_CFC_ (* Continuous Function Chart, elements in execution order *)
(* 3s *)
(* 3s *)
(* 90s *)
(* 1s *)
#0 AND(#3.Q, #6.Q)
#1 INT_TO_TIME(SHU6_PV1_ZADER_VPDS_OTSUT)
#2 MUL(#1, 1000)
#3 TON_PDS3:TON(IN: NOT SHU6_PV1_1PDS5_DI4, PT: #2)
#4 INT_TO_TIME(SHU6_PV1_ZADER_VPDS_RABOTA)
#5 MUL(#4, 1000)
#6 TON_ReRab:TON(IN: SHU6_PV1_UST_RE_RABOTA, PT: #5)
#7 INT_TO_TIME(SHU6_PV1_ZADER_M_VKL)
#8 MUL(#7, 1000)
#9 TON_MVKL_MV1:TON(IN: SHU6_PV1_MV1_DO3_VKL, PT: #8)
#10 INT_TO_TIME(SHU6_PV1_ZADER_M_A)
#11 MUL(#10, 1000)
#12 TON_AVT_MV1:TON(IN: SHU6_PV1_YAMV1_DI7_A, PT: #11)
#13 AND(#0, SHU6_PV1_MV1_B30, #9.Q, #12.Q)
#14 SR_NP_MV1:SR(SET1: #13, RESET: SHU6_PV1_SB)
#15 SHU6_PV1_Z_NETP_MV1 <= #14.Q1
_END_CFC_
(* the same logic as Structured Text *)
(* 3s *)
(* 3s *)
(* 90s *)
(* 1s *)
_t70 := TON_PDS3.Q AND TON_ReRab.Q;
TON_PDS3(IN := NOT SHU6_PV1_1PDS5_DI4, PT := INT_TO_TIME(SHU6_PV1_ZADER_VPDS_OTSUT) * 1000);
TON_ReRab(IN := SHU6_PV1_UST_RE_RABOTA, PT := INT_TO_TIME(SHU6_PV1_ZADER_VPDS_RABOTA) * 1000);
TON_MVKL_MV1(IN := SHU6_PV1_MV1_DO3_VKL, PT := INT_TO_TIME(SHU6_PV1_ZADER_M_VKL) * 1000);
TON_AVT_MV1(IN := SHU6_PV1_YAMV1_DI7_A, PT := INT_TO_TIME(SHU6_PV1_ZADER_M_A) * 1000);
SR_NP_MV1(SET1 := _t70 AND SHU6_PV1_MV1_B30 AND TON_MVKL_MV1.Q AND TON_AVT_MV1.Q, RESET := SHU6_PV1_SB);
SHU6_PV1_Z_NETP_MV1 := SR_NP_MV1.Q1;
END_PROGRAM

(* POU TZBiS/TZB/Z_NP_MRQ1, CFC *)
PROGRAM Z_NP_MRQ1
VAR
	SR_NP_M3: SR;
	TON_PDS1: TON;
	TON_ReRab: TON;
	TON_MVKL_M3: TON;
	TON_AVT_M3: TON;
END_VAR
VAR (* helpers for the ST form of the networks *)
	_t8 : TIME;
	_t13 : TIME;
	_t19 : TIME;
	_t25 : TIME;
	_t14 : TIME;
	_t20 : TIME;
	_t26 : TIME;
END_VAR
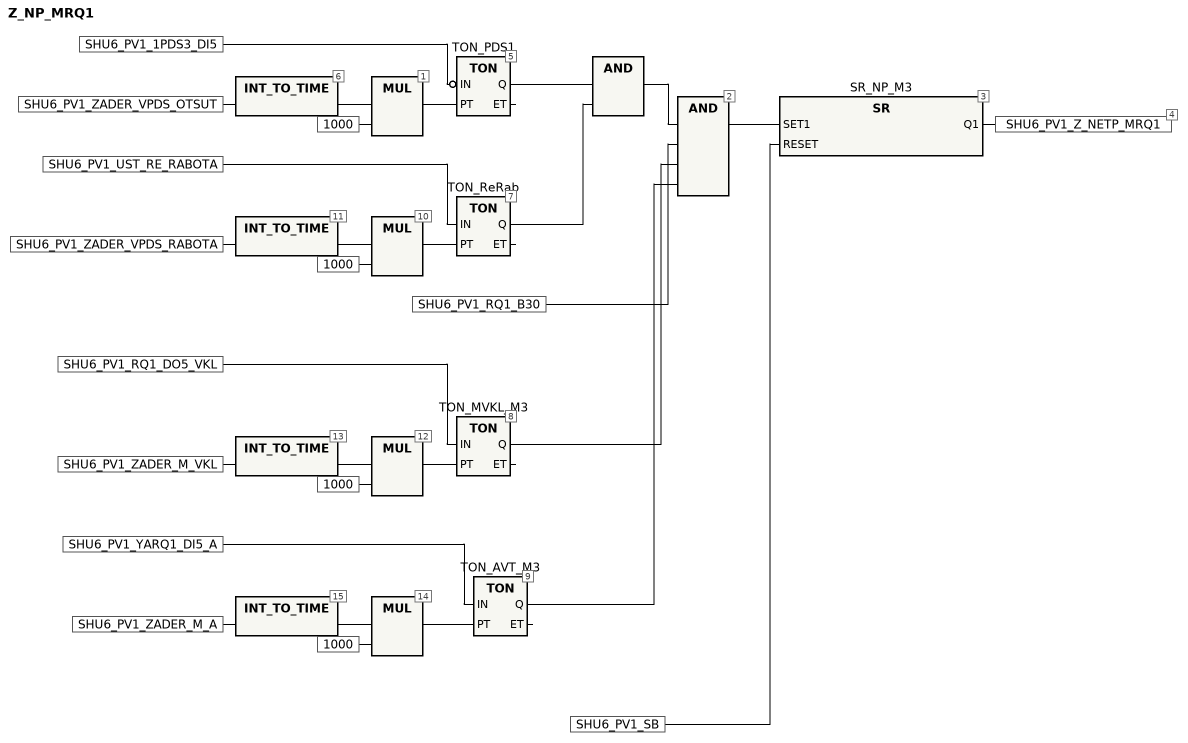
_CFC_ (* Continuous Function Chart, elements in execution order *)
#0 AND(#5.Q, #7.Q)
#1 MUL(#6, 1000)
#2 AND(#0, SHU6_PV1_RQ1_B30, #8.Q, #9.Q)
#3 SR_NP_M3:SR(SET1: #2, RESET: SHU6_PV1_SB)
#4 SHU6_PV1_Z_NETP_MRQ1 <= #3.Q1
#5 TON_PDS1:TON(IN: NOT SHU6_PV1_1PDS3_DI5, PT: #1)
#6 INT_TO_TIME(SHU6_PV1_ZADER_VPDS_OTSUT)
#7 TON_ReRab:TON(IN: SHU6_PV1_UST_RE_RABOTA, PT: #10)
#8 TON_MVKL_M3:TON(IN: SHU6_PV1_RQ1_DO5_VKL, PT: #12)
#9 TON_AVT_M3:TON(IN: SHU6_PV1_YARQ1_DI5_A, PT: #14)
#10 MUL(#11, 1000)
#11 INT_TO_TIME(SHU6_PV1_ZADER_VPDS_RABOTA)
#12 MUL(#13, 1000)
#13 INT_TO_TIME(SHU6_PV1_ZADER_M_VKL)
#14 MUL(#15, 1000)
#15 INT_TO_TIME(SHU6_PV1_ZADER_M_A)
_END_CFC_
(* the same logic as Structured Text *)
SR_NP_M3(SET1 := (TON_PDS1.Q AND TON_ReRab.Q) AND SHU6_PV1_RQ1_B30 AND TON_MVKL_M3.Q AND TON_AVT_M3.Q, RESET := SHU6_PV1_SB);
SHU6_PV1_Z_NETP_MRQ1 := SR_NP_M3.Q1;
TON_PDS1(IN := NOT SHU6_PV1_1PDS3_DI5, PT := _t8 * 1000);
_t8 := INT_TO_TIME(SHU6_PV1_ZADER_VPDS_OTSUT);
TON_ReRab(IN := SHU6_PV1_UST_RE_RABOTA, PT := _t13);
TON_MVKL_M3(IN := SHU6_PV1_RQ1_DO5_VKL, PT := _t19);
TON_AVT_M3(IN := SHU6_PV1_YARQ1_DI5_A, PT := _t25);
_t13 := _t14 * 1000;
_t14 := INT_TO_TIME(SHU6_PV1_ZADER_VPDS_RABOTA);
_t19 := _t20 * 1000;
_t20 := INT_TO_TIME(SHU6_PV1_ZADER_M_VKL);
_t25 := _t26 * 1000;
_t26 := INT_TO_TIME(SHU6_PV1_ZADER_M_A);
END_PROGRAM

(* POU TZBiS/TZB/Z_OTKAZ_VTOR_ZEP, CFC *)
PROGRAM Z_OTKAZ_VTOR_ZEP
VAR
	rs_otkaz_vtor_sep: RS;
	RS_102: RS;
	RS_QS: RS;
	RS_102_2: RS;
END_VAR
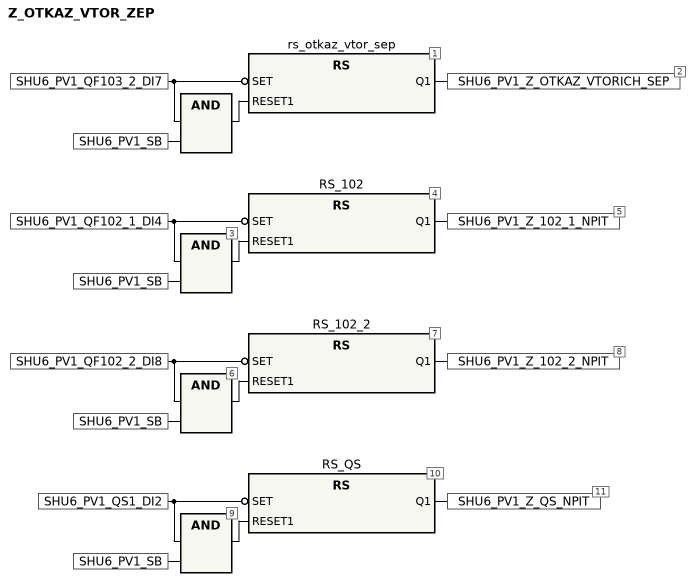
_CFC_ (* Continuous Function Chart, elements in execution order *)
#0 AND(SHU6_PV1_QF103_2_DI7, SHU6_PV1_SB)
#1 rs_otkaz_vtor_sep:RS(SET: NOT SHU6_PV1_QF103_2_DI7, RESET1: #0)
#2 SHU6_PV1_Z_OTKAZ_VTORICH_SEP <= #1.Q1
#3 AND(SHU6_PV1_QF102_1_DI4, SHU6_PV1_SB)
#4 RS_102:RS(SET: NOT SHU6_PV1_QF102_1_DI4, RESET1: #3)
#5 SHU6_PV1_Z_102_1_NPIT <= #4.Q1
#6 AND(SHU6_PV1_QF102_2_DI8, SHU6_PV1_SB)
#7 RS_102_2:RS(SET: NOT SHU6_PV1_QF102_2_DI8, RESET1: #6)
#8 SHU6_PV1_Z_102_2_NPIT <= #7.Q1
#9 AND(SHU6_PV1_QS1_DI2, SHU6_PV1_SB)
#10 RS_QS:RS(SET: NOT SHU6_PV1_QS1_DI2, RESET1: #9)
#11 SHU6_PV1_Z_QS_NPIT <= #10.Q1
_END_CFC_
(* the same logic as Structured Text *)
rs_otkaz_vtor_sep(SET := NOT SHU6_PV1_QF103_2_DI7, RESET1 := SHU6_PV1_QF103_2_DI7 AND SHU6_PV1_SB);
SHU6_PV1_Z_OTKAZ_VTORICH_SEP := rs_otkaz_vtor_sep.Q1;
RS_102(SET := NOT SHU6_PV1_QF102_1_DI4, RESET1 := SHU6_PV1_QF102_1_DI4 AND SHU6_PV1_SB);
SHU6_PV1_Z_102_1_NPIT := RS_102.Q1;
RS_102_2(SET := NOT SHU6_PV1_QF102_2_DI8, RESET1 := SHU6_PV1_QF102_2_DI8 AND SHU6_PV1_SB);
SHU6_PV1_Z_102_2_NPIT := RS_102_2.Q1;
RS_QS(SET := NOT SHU6_PV1_QS1_DI2, RESET1 := SHU6_PV1_QS1_DI2 AND SHU6_PV1_SB);
SHU6_PV1_Z_QS_NPIT := RS_QS.Q1;
END_PROGRAM

(* POU TZBiS/TZB/Z_P1_NP, CFC *)
PROGRAM Z_P1_NP
VAR
	SR_P1_NPit: SR;
END_VAR
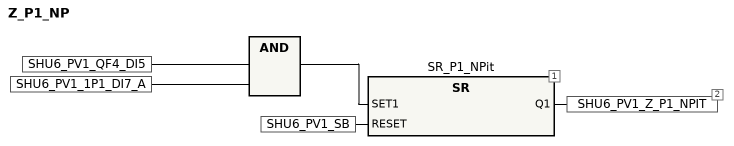
_CFC_ (* Continuous Function Chart, elements in execution order *)
#0 AND(SHU6_PV1_QF4_DI5, SHU6_PV1_1P1_DI7_A)
#1 SR_P1_NPit:SR(SET1: #0, RESET: SHU6_PV1_SB)
#2 SHU6_PV1_Z_P1_NPIT <= #1.Q1
_END_CFC_
(* the same logic as Structured Text *)
SR_P1_NPit(SET1 := SHU6_PV1_QF4_DI5 AND SHU6_PV1_1P1_DI7_A, RESET := SHU6_PV1_SB);
SHU6_PV1_Z_P1_NPIT := SR_P1_NPit.Q1;
END_PROGRAM

(* POU TZBiS/TZB/Sbros_All, CFC *)
PROGRAM Sbros_All
VAR
END_VAR
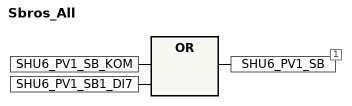
_CFC_ (* Continuous Function Chart, elements in execution order *)
#0 OR(SHU6_PV1_SB_KOM, SHU6_PV1_SB1_DI7)
#1 SHU6_PV1_SB <= #0
_END_CFC_
(* the same logic as Structured Text *)
SHU6_PV1_SB := SHU6_PV1_SB_KOM OR SHU6_PV1_SB1_DI7;
END_PROGRAM

(* POU TZBiS/TZB/Z_Pozhar, CFC *)
PROGRAM Z_Pozhar
VAR
	SR_Pozhar: SR;
END_VAR
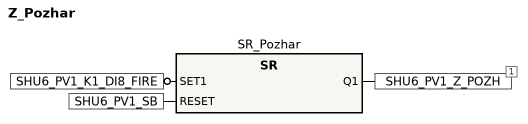
_CFC_ (* Continuous Function Chart, elements in execution order *)
#0 SR_Pozhar:SR(SET1: NOT SHU6_PV1_K1_DI8_FIRE, RESET: SHU6_PV1_SB)
#1 SHU6_PV1_Z_POZH <= #0.Q1
_END_CFC_
(* the same logic as Structured Text *)
SR_Pozhar(SET1 := NOT SHU6_PV1_K1_DI8_FIRE, RESET := SHU6_PV1_SB);
SHU6_PV1_Z_POZH := SR_Pozhar.Q1;
END_PROGRAM

(* POU TZBiS/TZB/Z_YA1_Otk, CFC *)
PROGRAM Z_YA1_Otk
VAR
	SR_YA1_OTKAZ: SR;
	TON_YA1_AVT: TON;
	TON_YA1_ZKR: TON;
	TON_YA1_OTKR: TON;
	TON_YA1_NE_OTKR: TON;
	TON_YA1_NE_ZAKR: TON;
END_VAR
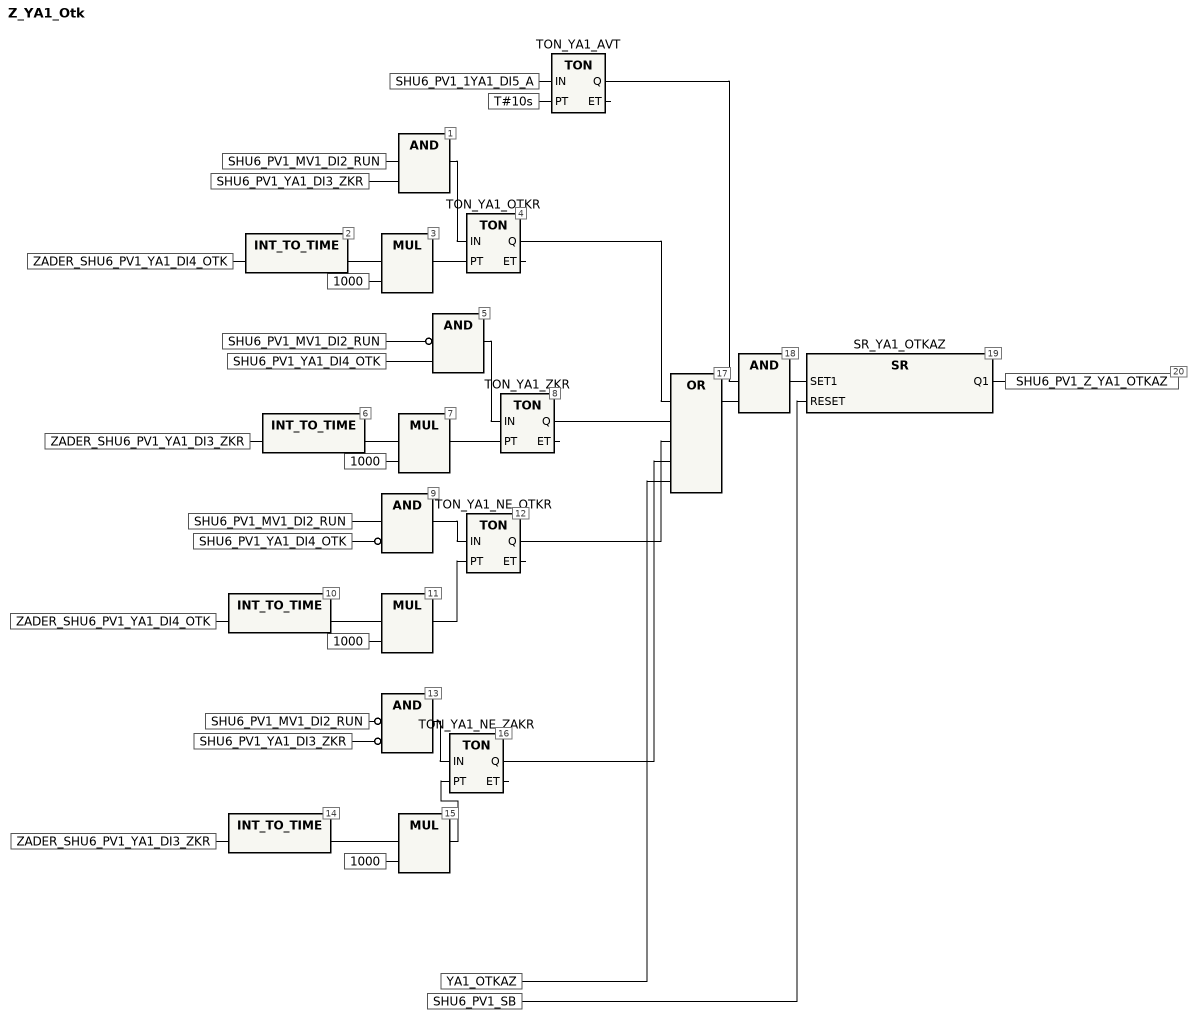
